// TIA Portal V18 export
FUNCTION_BLOCK "ConveyorFB"   // FB1, SCL
   VAR_INPUT
      StartPB : Bool;   // operator start pushbutton
      EStopOK : Bool;   // emergency stop healthy (safety)
      AutoMode : Bool;
      comm_err : Bool;
   END_VAR
   VAR_OUTPUT
      MotorRun : Bool;   // conveyor VFD run command
   END_VAR
   VAR
      ConvFault : Bool;
      vfd_err_timer : TON;
   END_VAR
BEGIN
   IF #StartPB AND #EStopOK AND #AutoMode AND NOT #ConvFault THEN
     #MotorRun := TRUE;
   END_IF;
   #vfd_err_timerIN := #comm_errPT := T#5S;
   IF #vfd_err_timer.Q THEN
     #ConvFault := TRUE;
   END_IF;
END_FUNCTION_BLOCK

VAR_GLOBAL   // PLC tag table "ConveyorTags"
   Motor_Out AT %Q0.0 : Bool;
   Start_In AT %I0.0 : Bool;
END_VAR
